FUNCTION_BLOCK EventToNumberAdapter_4
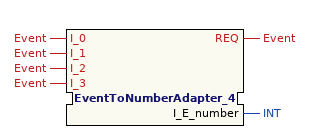
  EVENT_INPUT
    I_0;
    I_1;
    I_2;
    I_3;
  END_EVENT
  EVENT_OUTPUT
    REQ;
  END_EVENT
  VAR_OUTPUT
    I_E_number : INT;
  END_VAR
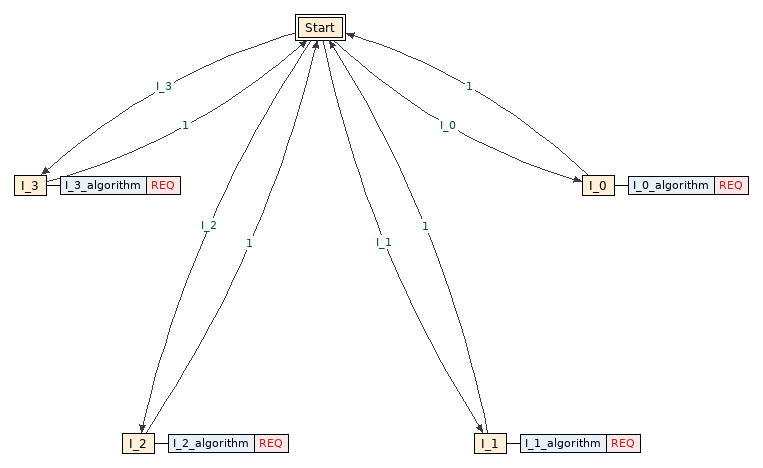
  EC_STATES
    Start;
    I_0 : I_0_algorithm -> REQ;
    I_1 : I_1_algorithm -> REQ;
    I_2 : I_2_algorithm -> REQ;
    I_3 : I_3_algorithm -> REQ;
  END_STATES
  EC_TRANSITIONS
    Start TO I_0 := I_0;
    I_0 TO Start := 1;
    Start TO I_1 := I_1;
    I_1 TO Start := 1;
    Start TO I_2 := I_2;
    I_2 TO Start := 1;
    Start TO I_3 := I_3;
    I_3 TO Start := 1;
  END_TRANSITIONS
  ALGORITHM I_0_algorithm IN ST:
I_E_number := 0;&#38;#10;
  END_ALGORITHM
  ALGORITHM I_1_algorithm IN ST:
I_E_number := 1;&#38;#10;
  END_ALGORITHM
  ALGORITHM I_2_algorithm IN ST:
I_E_number := 2;&#38;#10;
  END_ALGORITHM
  ALGORITHM I_3_algorithm IN ST:
I_E_number := 3;&#38;#10;
  END_ALGORITHM
END_FUNCTION_BLOCK
